# EPICS substitutions: ioc/morel/trunk/iocBoot/iocmorel/fb_epid.substitutions
# $Id: fb_epid.substitutions 14505 2012-02-29 21:25:07Z jemian $

file "$(OPTICS)/opticsApp/Db/fb_epid.db"
  {
    {
        P=morel:epid1,
	IN=morel:epid1:sim.VAL,
	OUT=morel:epid1:sim.D,
	MODE=PID,
	CALC=A,
	PERMIT1="morel:epid1:on.VAL",
	PERMIT2="",
	PERMIT3="",
	PERMIT4=""
    }
  }
